{attribute 'no_explicit_call' := 'do not call this function block directly'} 
PROGRAM ExceptionManager
VAR
	_Exception : POINTER TO Exception;
	_EmptyException : EmptyException;
	_SystemException : SystemException;	
END_VAR

METHOD Cleanup
IF _Exception <> 0 THEN
	__DELETE(_Exception);		
END_IF
END_METHOD

// Result is always not null. Returns EmptyException instance by default
METHOD GetLastException : IException
VAR_IN_OUT CONSTANT 
	exceptionCode : __SYSTEM.ExceptionCode;
END_VAR
IF exceptionCode = __SYSTEM.ExceptionCode.RTSEXCPT_DIVIDEBYZERO AND_THEN _Exception <> 0 THEN
	GetLastException := _Exception^;
ELSE
	_SystemException.SetExceptionCode(exceptionCode);
	GetLastException := _SystemException;
END_IF
END_METHOD

METHOD Throw
VAR_INPUT
	exception : IException;
END_VAR
VAR
	fakeVariable : INT := 0;
	exceptionCloneInterface : IObject;
END_VAR
IF _Exception <> 0 THEN
	__DELETE(_Exception);
END_IF

__QUERYPOINTER(exception.Clone(), _Exception);

// fake devision by zero
fakeVariable := fakeVariable / fakeVariable;
END_METHOD

END_PROGRAM

(* stored: Version 1.1.0.1
   POU ExceptionManager: Id {722e8a75-a8dc-4f6d-84e9-83f307045e70}, SpecialFunc None
   Method Cleanup: Id {f9d00147-ef5a-438a-91f3-6814363f412d}
   Method GetLastException: Id {434a5e87-4296-4bc5-a3c7-e1fd25672e22}
   Method Throw: Id {749562e1-1a92-4b62-b485-e35611af487a} *)
